
FUNCTION CB_word_to_real : REAL


TITLE = ' Convert an word into a real '
VERSION : '1.0'
AUTHOR  : CB
NAME    : wordToRe
FAMILY  : TNI

VAR_INPUT
    IN : WORD;
END_VAR

BEGIN
CB_word_to_real := DINT_TO_REAL(WORD_TO_DINT(IN));

END_FUNCTION
